METHOD CamAddPointToPath : BOOL
VAR_INPUT
	MotionFunctionFirstPoint : MC_MotionFunctionType;										  // Motion Function Type of initial Point in Cam Table. Start Postion is defined by current Positon of Axes.
	MotionFunctionThisPoint	 : MC_MotionFunctionType;										  // Motion Function Type of this Point to be added to Cam-Table
	PointNumber				 : UDINT(2..Parameter_Kinematic.MaxCammingPositionsPerTable);	  // Number of Point to be added to Cam Table, must be strictly increasing without gaps
	TotalPointsInTable		 : UDINT(2..Parameter_Kinematic.MaxCammingPositionsPerTable);	  // Total Number of Points in final Cam Table
	PointVelocity			 : ARRAY[1..KINEMATIC_CONSTANTS.DEGREES_OF_FREEDOM_MAX] OF LREAL; // Slave Velocity at this Point in Cam Table
	PointAcceleration		 : ARRAY[1..KINEMATIC_CONSTANTS.DEGREES_OF_FREEDOM_MAX] OF LREAL; // Slave Acceleration at this Point in Cam Table
	PointJerk				 : ARRAY[1..KINEMATIC_CONSTANTS.DEGREES_OF_FREEDOM_MAX] OF LREAL; // Slave Jerk at this Point in Cam Table
	PointIndex				 : UDINT;														  // Index of Point in structure of ST_BasePoint
END_VAR
IF _AcsAxesCam.CammingActive OR _McsAxesCam.CammingActive OR _AcsAxesCam.Busy OR _McsAxesCam.Busy THEN
	TRACE('CamAddPointToPath - Camming active or Buys');
	RETURN;
END_IF

IF SUPER^.KinematicStatus = E_KinStatus.KinStatus_Empty THEN
	CamAddPointToPath := _AcsAxesCam.CamAddPointToPath(MotionFunctionFirstPoint := MotionFunctionFirstPoint,
													   MotionFunctionThisPoint	:= MotionFunctionThisPoint,
													   PointNumber				:= PointNumber,
													   TotalPointsInTable		:= TotalPointsInTable,
													   Point					:= _CamPoints[PointIndex].AcsPosition,
													   PointVelocity			:= PointVelocity,
													   PointAcceleration		:= PointAcceleration,
													   PointJerk				:= PointJerk);
ELSIF SUPER^.KinematicStatus = E_KinStatus.KinStatus_Ready THEN
	CamAddPointToPath := _McsAxesCam.CamAddPointToPath(MotionFunctionFirstPoint := MotionFunctionFirstPoint,
													   MotionFunctionThisPoint	:= MotionFunctionThisPoint,
													   PointNumber				:= PointNumber,
													   TotalPointsInTable		:= TotalPointsInTable,
													   Point					:= _CamPoints[PointIndex].McsPosition,
													   PointVelocity			:= PointVelocity,
													   PointAcceleration		:= PointAcceleration,
													   PointJerk				:= PointJerk);
ELSE
	CamAddPointToPath := FALSE;
END_IF
END_METHOD

PROPERTY PUBLIC ChangeOccurred : BOOL
GET
ChangeOccurred := _ChangeOccurred;
END_GET
SET
_ChangeOccurred := ChangeOccurred;
END_SET
END_PROPERTY

METHOD PUBLIC GetPoint : ST_BasePoint
VAR_INPUT
	PointIndex : UDINT;
END_VAR
IF PointIndex > Parameter_Kinematic.MaxPoints THEN
	RETURN;
END_IF

GetPoint := _CamPoints[PointIndex];
END_METHOD

PROPERTY Points : REFERENCE TO ARRAY[0..Parameter_Kinematic.MaxPoints] OF ST_BasePoint
GET
Points REF= _CamPoints;
END_GET
END_PROPERTY

METHOD PUBLIC SetPoint : BOOL
VAR_INPUT
	Point	   : ST_BasePoint;
	PointIndex : UDINT;
END_VAR
IF PointIndex > Parameter_Kinematic.MaxPoints THEN
	RETURN;
END_IF

_CamPoints[PointIndex] := Point;
_ChangeOccurred		   := TRUE;
SetPoint			   := TRUE;
END_METHOD

PROPERTY CamInOptionsACS : ST_CamInOptions
GET
CamInOptionsACS := _AcsAxesCam.CamInOptions;
END_GET
SET
_AcsAxesCam.CamInOptions := CamInOptionsACS;
END_SET
END_PROPERTY

PROPERTY CamInOptionsMCS : ST_CamInOptions
GET
CamInOptionsMCS := _MCSAxesCam.CamInOptions;
END_GET
SET
_MCSAxesCam.CamInOptions := CamInOptionsMCS;
END_SET
END_PROPERTY

PROPERTY CamMasterAcs : REFERENCE TO AXIS_REF
GET
CamMasterAcs REF= _AcsAxesCam.CamMaster;
END_GET
END_PROPERTY

PROPERTY CamMasterMcs : REFERENCE TO AXIS_REF
GET
CamMasterMcs REF= _McsAxesCam.CamMaster;
END_GET
END_PROPERTY

PROPERTY CamTableSlaveDynamicsACS : ARRAY[1..KINEMATIC_CONSTANTS.DEGREES_OF_FREEDOM_MAX] OF ST_CamTableSlaveDynamics;
GET
CamTableSlaveDynamicsACS := _AcsAxesCam.CamTableSlaveDynamics;
END_GET
END_PROPERTY

PROPERTY CamTableSlaveDynamicsMCS : ARRAY[1..KINEMATIC_CONSTANTS.DEGREES_OF_FREEDOM_MAX] OF ST_CamTableSlaveDynamics;
GET
CamTableSlaveDynamicsMCS := _McsAxesCam.CamTableSlaveDynamics;
END_GET
END_PROPERTY

//! @summary Basic component initialization logic
METHOD PROTECTED Initialize : BOOL;
_AcsAxesCam.CamAxisCount := TO_UDINT(iAxis.AcsAxisCount);
_AcsAxesCam.CamAxisRef	 REF= iAxis.ACS;
_McsAxesCam.CamAxisCount := TO_UDINT(iAxis.DegreesOfFreedomConfigured);
_McsAxesCam.CamAxisRef	 REF= iAxis.MCS;
_AcsAxesCam.CyclicLogic(); // Init Run
_McsAxesCam.CyclicLogic(); // Init Run
IF SUPER^.Initialize() THEN
	Initialize := _AcsAxesCam.InitComplete AND _McsAxesCam.InitComplete;
END_IF
END_METHOD

END_FUNCTION_BLOCK

// Interfaces/I_KinematicCamming
INTERFACE I_KinematicCamming

METHOD CamClearPath : BOOL
VAR_INPUT
END_VAR
END_METHOD

METHOD CamIn : BOOL
VAR_INPUT
END_VAR
END_METHOD

METHOD CamMasterZero : BOOL
VAR_INPUT
END_VAR
END_METHOD

METHOD CamOut : BOOL
VAR_INPUT
END_VAR
END_METHOD

METHOD CamStartMovePath : BOOL
VAR_INPUT
	TargetMoveVelocity	   : LREAL := Parameter_Kinematic.CamDefaultMoveVelocity;	  // Move Velocity for Cam Table Master !!!Needs to consider all Slave dynamics, all Slaves try to follow Master setpoints!!!
	TargetMoveAcceleration : LREAL := Parameter_Kinematic.CamDefaultMoveAcceleration; // Move Acceleration for Cam Table Master !!!Needs to consider all Slave dynamics, all Slaves try to follow Master setpoints!!!
	TargetMoveDeceleration : LREAL := Parameter_Kinematic.CamDefaultMoveDeceleration; // Move Deceleration for Cam Table Master !!!Needs to consider all Slave dynamics, all Slaves try to follow Master setpoints!!!
	TargetMoveJerk		   : LREAL := Parameter_Kinematic.CamDefaultMoveJerk;		  // Move Jerk for Cam Table Master !!!Needs to consider all Slave dynamics, all Slaves try to follow Master setpoints!!!
END_VAR
END_METHOD

PROPERTY CammingActive : BOOL
GET
END_GET
END_PROPERTY

END_INTERFACE

// FunctionBlocks/FB_KinematicCamming
FUNCTION_BLOCK FB_KinematicCamming EXTENDS FB_CyclicFB IMPLEMENTS I_KinematicCamming
VAR
	// Kinematic Axis
	_CamVirtualMaster	  : AXIS_REF;
	_CamAxisRef			  : REFERENCE TO ARRAY[1..KINEMATIC_CONSTANTS.DEGREES_OF_FREEDOM_MAX] OF AXIS_REF;
	_CamAxisCount		  : UDINT := 1;
	_MotionFunctionPoints : ARRAY[1..KINEMATIC_CONSTANTS.DEGREES_OF_FREEDOM_MAX] OF UDINT(2..Parameter_Kinematic.MaxCammingPositionsPerTable) := [2,2,2,2,2,2];

	// Camming
	_McCamTableSelect		     : ARRAY[1..KINEMATIC_CONSTANTS.DEGREES_OF_FREEDOM_MAX] OF MC_CamTableSelect;
	_TableCamRef			     : ARRAY[1..KINEMATIC_CONSTANTS.DEGREES_OF_FREEDOM_MAX] OF MC_CAM_REF;
	_MotionFunctionPointsAxis1   : ARRAY[1..Parameter_Kinematic.MaxCammingPositionsPerTable] OF MC_MotionFunctionPoint;
	_MotionFunctionPointsAxis2   : ARRAY[1..Parameter_Kinematic.MaxCammingPositionsPerTable] OF MC_MotionFunctionPoint;
	_MotionFunctionPointsAxis3   : ARRAY[1..Parameter_Kinematic.MaxCammingPositionsPerTable] OF MC_MotionFunctionPoint;
	_MotionFunctionPointsAxis4   : ARRAY[1..Parameter_Kinematic.MaxCammingPositionsPerTable] OF MC_MotionFunctionPoint;
	_MotionFunctionPointsAxis5   : ARRAY[1..Parameter_Kinematic.MaxCammingPositionsPerTable] OF MC_MotionFunctionPoint;
	_MotionFunctionPointsAxis6   : ARRAY[1..Parameter_Kinematic.MaxCammingPositionsPerTable] OF MC_MotionFunctionPoint;
	_McCamIn				     : ARRAY[1..KINEMATIC_CONSTANTS.DEGREES_OF_FREEDOM_MAX] OF MC_CamIn;
	_McCamOut				     : ARRAY[1..KINEMATIC_CONSTANTS.DEGREES_OF_FREEDOM_MAX] OF MC_CamOut;
	_McReadCamTableSlaveDynamics : ARRAY[1..KINEMATIC_CONSTANTS.DEGREES_OF_FREEDOM_MAX] OF MC_ReadCamTableSlaveDynamics;
	_CamTableSlaveDynamics       : ARRAY[1..KINEMATIC_CONSTANTS.DEGREES_OF_FREEDOM_MAX] OF ST_CamTableSlaveDynamics;
	_McPowerVirtualMaster	     : MC_POWER;
	_McMoveAbs				     : MC_MoveAbsolute;
	_McHalt					     : MC_Halt;
	_McReset				     : MC_Reset;
	_McHome					     : MC_HOME;
	_CamInOptions                : ST_CamInOptions;

	// Internal Variables
	_KinematicCamInit		  : E_InitializeState_KinematicCamming := E_InitializeState_KinematicCamming.eInitializeState_Start;
	_i						  : UDINT;
	_MotionFunctionFirstPoint : MC_MotionFunctionType := MC_MotionFunctionType.MOTIONFUNCTYPE_POLYNOM5;
END_VAR

METHOD PUBLIC CyclicLogic
IF NOT _InitComplete THEN
	_InitComplete := THIS^.Initialize();
	RETURN;
END_IF

_CamVirtualMaster.ReadStatus();

(* Power Virtual Master *)
_McPowerVirtualMaster(Axis := _CamVirtualMaster, Enable_Positive := TRUE, Enable_Negative := TRUE);
IF _McPowerVirtualMaster.Error THEN
	_Error	 := TRUE;
	_ErrorId := _McPowerVirtualMaster.ErrorID;
END_IF

(* Reset Virtual Master *)
_McReset(Axis := _CamVirtualMaster);
IF _McReset.Error THEN
	_Error	 := TRUE;
	_ErrorId := _McReset.ErrorID;
END_IF

_McReset.Execute := FALSE;

(* Stop Virtual Master *)
_McHalt(Axis := _CamVirtualMaster);
IF _McHalt.Error THEN
	_Error	 := TRUE;
	_ErrorId := _McHalt.ErrorID;
END_IF

_McHalt.Execute := FALSE;

(* Move Virtual Master *)
_McMoveAbs(Axis := _CamVirtualMaster);
IF _McMoveAbs.Error THEN
	_Error	 := TRUE;
	_ErrorId := _McMoveAbs.ErrorID;
END_IF

_McMoveAbs.Execute := FALSE;

(* Reset Master to 0 *)
_McHome(Axis := _CamVirtualMaster, Position := 0.0, HomingMode := MC_HomingMOde.MC_Direct);
IF _McHome.Error THEN
	_Error	 := TRUE;
	_ErrorId := _McHome.ErrorID;
END_IF

_McHome.Execute := FALSE;

(* Reference Cam Table and initate first point *)
_TableCamRef[1].pArray		:= ADR(_MotionFunctionPointsAxis1);
_TableCamRef[1].ArraySize	:= SIZEOF(_MotionFunctionPointsAxis1);
_TableCamRef[1].TableType	:= MC_TableType.MC_TABLETYPE_MOTIONFUNCTION;
_TableCamRef[1].NoOfColumns := 1;
_TableCamRef[1].NoOfRows	:= _MotionFunctionPoints[1];
_TableCamRef[2].pArray		:= ADR(_MotionFunctionPointsAxis2);
_TableCamRef[2].ArraySize	:= SIZEOF(_MotionFunctionPointsAxis2);
_TableCamRef[2].TableType	:= MC_TableType.MC_TABLETYPE_MOTIONFUNCTION;
_TableCamRef[2].NoOfColumns := 1;
_TableCamRef[2].NoOfRows	:= _MotionFunctionPoints[2];
_TableCamRef[3].pArray		:= ADR(_MotionFunctionPointsAxis3);
_TableCamRef[3].ArraySize	:= SIZEOF(_MotionFunctionPointsAxis3);
_TableCamRef[3].TableType	:= MC_TableType.MC_TABLETYPE_MOTIONFUNCTION;
_TableCamRef[3].NoOfColumns := 1;
_TableCamRef[3].NoOfRows	:= _MotionFunctionPoints[3];
_TableCamRef[4].pArray		:= ADR(_MotionFunctionPointsAxis4);
_TableCamRef[4].ArraySize	:= SIZEOF(_MotionFunctionPointsAxis4);
_TableCamRef[4].TableType	:= MC_TableType.MC_TABLETYPE_MOTIONFUNCTION;
_TableCamRef[4].NoOfColumns := 1;
_TableCamRef[4].NoOfRows	:= _MotionFunctionPoints[4];
_TableCamRef[5].pArray		:= ADR(_MotionFunctionPointsAxis5);
_TableCamRef[5].ArraySize	:= SIZEOF(_MotionFunctionPointsAxis5);
_TableCamRef[5].TableType	:= MC_TableType.MC_TABLETYPE_MOTIONFUNCTION;
_TableCamRef[5].NoOfColumns := 1;
_TableCamRef[5].NoOfRows	:= _MotionFunctionPoints[5];
_TableCamRef[6].pArray		:= ADR(_MotionFunctionPointsAxis6);
_TableCamRef[6].ArraySize	:= SIZEOF(_MotionFunctionPointsAxis6);
_TableCamRef[6].TableType	:= MC_TableType.MC_TABLETYPE_MOTIONFUNCTION;
_TableCamRef[6].NoOfColumns := 1;
_TableCamRef[6].NoOfRows	:= _MotionFunctionPoints[6];
FOR _i := 1 TO _CamAxisCount DO
	(* Build Cam Table *)
	_McCamTableSelect[_i](Master		 := _CamVirtualMaster,
						  Slave			 := _CamAxisRef[_i],
						  CamTable		 := _TableCamRef[_i],
						  Periodic		 := Parameter_Kinematic.ExecuteCamPeriodically,
						  MasterAbsolute := Parameter_Kinematic.CamMasterAbsolute,
						  SlaveAbsolute	 := Parameter_Kinematic.CamSlaveAbsolute,
						  CamTableId	 := (_CamAxisRef[_i].NcToPlc.AxisId * 100));

	IF _McCamTableSelect[_i].Error THEN
		_Error	 := TRUE;
		_ErrorId := _McCamTableSelect[_i].ErrorID;
	END_IF

	_McCamTableSelect[_i].Execute := FALSE;

	(* Cam Axes to Master *)
	_McCamIn[_i](Master		   := _CamVirtualMaster,
				 Slave		   := _CamAxisRef[_i],
				 MasterOffset  := 0,
				 SlaveOffset   := 0,
				 MasterScaling := 1,
				 SlaveScaling  := 1,
				 StartMode	   := MC_STARTMODE.MC_STARTMODE_ABSOLUTE,
				 CamTableId	   := (_CamAxisRef[_i].NcToPlc.AxisId * 100),
				 Options	   := _CamInOptions);

	IF _McCamIn[_i].Error THEN
		_Error	 := TRUE;
		_ErrorId := _McCamIn[_i].ErrorID;
	END_IF

	_McCamIn[_i].Execute := FALSE;

	(* Cam Out Axes to Master *)
	_McCamOut[_i](Slave := _CamAxisRef[_i]);
	IF _McCamOut[_i].Error THEN
		_Error	 := TRUE;
		_ErrorId := _McCamOut[_i].ErrorID;
	END_IF

	_McCamOut[_i].Execute := FALSE;

	(* MC_ReadCamTableSlaveDynamics *)
	_McReadCamTableSlaveDynamics[_i](CamTableId		   := (_CamAxisRef[_i].NcToPlc.AxisId * 100),
									 SlavePosition	   => _CamTableSlaveDynamics[_i].SlavePosition,
									 SlaveVelocity	   => _CamTableSlaveDynamics[_i].SlaveVelocity,
									 SlaveAcceleration => _CamTableSlaveDynamics[_i].SlaveAcceleration);

	_McReadCamTableSlaveDynamics[_i].Execute := FALSE;
END_FOR

(* Create Busy Signal *)
_Busy := _McHalt.Busy OR _McReset.Busy OR _McMoveAbs.Busy OR _McHome.Busy;
FOR _i := 1 TO _CamAxisCount DO
	IF _McCamIn[_i].Busy OR _McCamOut[_i].Busy OR _McCamTableSelect[_i].Busy OR _McReadCamTableSlaveDynamics[_i].Busy THEN
		_Busy := TRUE;
	END_IF
END_FOR
END_METHOD

METHOD CamClearPath : BOOL
IF _Busy OR CammingActive THEN
	RETURN;
END_IF

MEMSET(destAddr := ADR(_MotionFunctionPointsAxis1), fillByte := 0, n := SIZEOF(_MotionFunctionPointsAxis1));
MEMSET(destAddr := ADR(_MotionFunctionPointsAxis2), fillByte := 0, n := SIZEOF(_MotionFunctionPointsAxis2));
MEMSET(destAddr := ADR(_MotionFunctionPointsAxis3), fillByte := 0, n := SIZEOF(_MotionFunctionPointsAxis3));
MEMSET(destAddr := ADR(_MotionFunctionPointsAxis4), fillByte := 0, n := SIZEOF(_MotionFunctionPointsAxis4));
MEMSET(destAddr := ADR(_MotionFunctionPointsAxis5), fillByte := 0, n := SIZEOF(_MotionFunctionPointsAxis5));
MEMSET(destAddr := ADR(_MotionFunctionPointsAxis6), fillByte := 0, n := SIZEOF(_MotionFunctionPointsAxis6));
CamClearPath := TRUE;
END_METHOD

METHOD CamIn : BOOL
IF _Busy OR CammingActive THEN
	RETURN;
END_IF

FOR _i := 1 TO _CamAxisCount DO
	_McCamIn[_i].Execute := TRUE;
END_FOR

CamIn := TRUE;
END_METHOD

METHOD CamMasterZero : BOOL
VAR_INPUT
END_VAR
IF _Busy OR CammingActive THEN
	RETURN;
END_IF

_McHome.Execute := TRUE;
CamMasterZero	:= TRUE;
END_METHOD

{attribute 'monitoring' := 'variable'}
PROPERTY CammingActive : BOOL
GET
CammingActive := TRUE;
FOR _i := 1 TO _CamAxisCount DO
	IF _CamAxisRef[_i].NcToPlc.CoupleState <> 3 THEN
		CammingActive := False;
	END_IF
END_FOR
END_GET
END_PROPERTY

METHOD CamOut : BOOL
IF _Busy THEN
	RETURN;
END_IF

FOR _i := 1 TO _CamAxisCount DO
	_McCamOut[_i].Execute := TRUE;
END_FOR

CamOut := TRUE;
END_METHOD

METHOD CamStartMovePath : BOOL
VAR_INPUT
	TargetMoveVelocity	   : LREAL := Parameter_Kinematic.CamDefaultMoveVelocity;	  // Move Velocity for Cam Table Master !!!Needs to consider all Slave dynamics, all Slaves try to follow Master setpoints!!!
	TargetMoveAcceleration : LREAL := Parameter_Kinematic.CamDefaultMoveAcceleration; // Move Acceleration for Cam Table Master !!!Needs to consider all Slave dynamics, all Slaves try to follow Master setpoints!!!
	TargetMoveDeceleration : LREAL := Parameter_Kinematic.CamDefaultMoveDeceleration; // Move Deceleration for Cam Table Master !!!Needs to consider all Slave dynamics, all Slaves try to follow Master setpoints!!!
	TargetMoveJerk		   : LREAL := Parameter_Kinematic.CamDefaultMoveJerk;		  // Move Jerk for Cam Table Master !!!Needs to consider all Slave dynamics, all Slaves try to follow Master setpoints!!!
END_VAR
IF _Busy OR NOT CammingActive THEN
	RETURN;
END_IF

_McMoveAbs.Jerk			:= TargetMoveJerk;
_McMoveAbs.Acceleration := TargetMoveAcceleration;
_McMoveAbs.Deceleration := TargetMoveDeceleration;
_McMoveAbs.Velocity		:= TargetMoveVelocity;
_McMoveAbs.Position		:= _CamVirtualMaster.NcToPlc.ActPos + 1.0;
_McMoveAbs.Execute		:= TRUE;
CamStartMovePath		:= TRUE;
END_METHOD

METHOD CamAddMotionPointByAxis : BOOL
VAR_INPUT
	Axis					 : UDINT(1..KINEMATIC_CONSTANTS.DEGREES_OF_FREEDOM_MAX);				   // Axis Number to add point to Cam table
	MotionFunctionFirstPoint : MC_MotionFunctionType := MC_MotionFunctionType.MOTIONFUNCTYPE_POLYNOM5; // Motion Function Type of initial Point in Cam Table. Start Postion is defined by current Positon of Axes.
	MotionFunctionThisPoint	 : MC_MotionFunctionType := MC_MotionFunctionType.MOTIONFUNCTYPE_POLYNOM5; // Motion Function Type of this Point to be added to Cam-Table
	PointNumber				 : UDINT(1..Parameter_Kinematic.MaxCammingPositionsPerTable);			   // Number of Point to be added to Cam Table, must be strictly increasing without gaps
	TotalPointsInTable		 : UDINT(2..Parameter_Kinematic.MaxCammingPositionsPerTable);			   // Total Number of Points in final Cam Table
	MasterPosition			 : LREAL;																   // Master Position for this Motion Point scaled to 1
	SlavePosition			 : LREAL;																   // Slave Position at this Point in Cam Table
	PointVelocity			 : LREAL;																   // Slave Velocity at this Point in Cam Table
	PointAcceleration		 : LREAL;																   // Slave Acceleration at this Point in Cam Table
	PointJerk				 : LREAL;																   // Slave Jerk at this Point in Cam Table
END_VAR

VAR
	_NextRelPoint : UDINT;
END_VAR
IF _Busy OR CammingActive THEN
	TRACE('CamAddMotionPointByAxis - Rejected buys or camming active!');
	RETURN;
END_IF

IF PointNumber > TotalPointsInTable OR PointNumber > Parameter_Kinematic.MaxCammingPositionsPerTable THEN
	TRACE('CamAddMotionPointByAxis - Rejected PointNumber invalid!');
	RETURN;
END_IF

IF MasterPosition < 0.0 OR MasterPosition > 1.0 THEN
	TRACE('CamAddMotionPointByAxis - Rejected MasterPosition not in allowed range of 0.0..1.0!');
	RETURN;
END_IF

IF NOT Parameter_Kinematic.CammingFirstPointInTableByUser THEN
	CamTableAddStartPoint();
END_IF

CASE Axis OF
	1:
		_MotionFunctionFirstPoint := MotionFunctionFirstPoint;
		IF PointNumber = TotalPointsInTable THEN
			_NextRelPoint				 := 0;
			_MotionFunctionPoints[1]	 := TotalPointsInTable;
			_McCamTableSelect[1].Execute := TRUE;
		ELSE
			_NextRelPoint := 1;
		END_IF

		_MotionFunctionPointsAxis1[PointNumber].PointIndex		  := PointNumber;
		_MotionFunctionPointsAxis1[PointNumber].FunctionType	  := MotionFunctionThisPoint;
		_MotionFunctionPointsAxis1[PointNumber].PointType		  := MC_MotionPointType.MOTIONPOINTTYPE_MOTION;
		_MotionFunctionPointsAxis1[PointNumber].MasterPos		  := MasterPosition;
		_MotionFunctionPointsAxis1[PointNumber].RelIndexNextPoint := _NextRelPoint;
		_MotionFunctionPointsAxis1[PointNumber].SlavePos		  := SlavePosition;
		_MotionFunctionPointsAxis1[PointNumber].SlaveVelo		  := PointVelocity;
		_MotionFunctionPointsAxis1[PointNumber].SlaveAcc		  := PointAcceleration;
		_MotionFunctionPointsAxis1[PointNumber].SlaveJerk		  := PointJerk;
		CamAddMotionPointByAxis									  := TRUE;

	2:
		_MotionFunctionFirstPoint := MotionFunctionFirstPoint;
		IF PointNumber = TotalPointsInTable THEN
			_NextRelPoint				 := 0;
			_MotionFunctionPoints[2]	 := TotalPointsInTable;
			_McCamTableSelect[2].Execute := TRUE;
		ELSE
			_NextRelPoint := 1;
		END_IF

		_MotionFunctionPointsAxis2[PointNumber].PointIndex		  := PointNumber;
		_MotionFunctionPointsAxis2[PointNumber].FunctionType	  := MotionFunctionThisPoint;
		_MotionFunctionPointsAxis2[PointNumber].PointType		  := MC_MotionPointType.MOTIONPOINTTYPE_MOTION;
		_MotionFunctionPointsAxis2[PointNumber].MasterPos		  := MasterPosition;
		_MotionFunctionPointsAxis2[PointNumber].RelIndexNextPoint := _NextRelPoint;
		_MotionFunctionPointsAxis2[PointNumber].SlavePos		  := SlavePosition;
		_MotionFunctionPointsAxis2[PointNumber].SlaveVelo		  := PointVelocity;
		_MotionFunctionPointsAxis2[PointNumber].SlaveAcc		  := PointAcceleration;
		_MotionFunctionPointsAxis2[PointNumber].SlaveJerk		  := PointJerk;
		CamAddMotionPointByAxis									  := TRUE;

	3:
		_MotionFunctionFirstPoint := MotionFunctionFirstPoint;
		IF PointNumber = TotalPointsInTable THEN
			_NextRelPoint				 := 0;
			_MotionFunctionPoints[3]	 := TotalPointsInTable;
			_McCamTableSelect[3].Execute := TRUE;
		ELSE
			_NextRelPoint := 1;
		END_IF

		_MotionFunctionPointsAxis3[PointNumber].PointIndex		  := PointNumber;
		_MotionFunctionPointsAxis3[PointNumber].FunctionType	  := MotionFunctionThisPoint;
		_MotionFunctionPointsAxis3[PointNumber].PointType		  := MC_MotionPointType.MOTIONPOINTTYPE_MOTION;
		_MotionFunctionPointsAxis3[PointNumber].MasterPos		  := MasterPosition;
		_MotionFunctionPointsAxis3[PointNumber].RelIndexNextPoint := _NextRelPoint;
		_MotionFunctionPointsAxis3[PointNumber].SlavePos		  := SlavePosition;
		_MotionFunctionPointsAxis3[PointNumber].SlaveVelo		  := PointVelocity;
		_MotionFunctionPointsAxis3[PointNumber].SlaveAcc		  := PointAcceleration;
		_MotionFunctionPointsAxis3[PointNumber].SlaveJerk		  := PointJerk;
		CamAddMotionPointByAxis									  := TRUE;

	4:
		_MotionFunctionFirstPoint := MotionFunctionFirstPoint;
		IF PointNumber = TotalPointsInTable THEN
			_NextRelPoint				 := 0;
			_MotionFunctionPoints[4]	 := TotalPointsInTable;
			_McCamTableSelect[4].Execute := TRUE;
		ELSE
			_NextRelPoint := 1;
		END_IF

		_MotionFunctionPointsAxis4[PointNumber].PointIndex		  := PointNumber;
		_MotionFunctionPointsAxis4[PointNumber].FunctionType	  := MotionFunctionThisPoint;
		_MotionFunctionPointsAxis4[PointNumber].PointType		  := MC_MotionPointType.MOTIONPOINTTYPE_MOTION;
		_MotionFunctionPointsAxis4[PointNumber].MasterPos		  := MasterPosition;
		_MotionFunctionPointsAxis4[PointNumber].RelIndexNextPoint := _NextRelPoint;
		_MotionFunctionPointsAxis4[PointNumber].SlavePos		  := SlavePosition;
		_MotionFunctionPointsAxis4[PointNumber].SlaveVelo		  := PointVelocity;
		_MotionFunctionPointsAxis4[PointNumber].SlaveAcc		  := PointAcceleration;
		_MotionFunctionPointsAxis4[PointNumber].SlaveJerk		  := PointJerk;
		CamAddMotionPointByAxis									  := TRUE;

	5:
		_MotionFunctionFirstPoint := MotionFunctionFirstPoint;
		IF PointNumber = TotalPointsInTable THEN
			_NextRelPoint				 := 0;
			_MotionFunctionPoints[5]	 := TotalPointsInTable;
			_McCamTableSelect[5].Execute := TRUE;
		ELSE
			_NextRelPoint := 1;
		END_IF

		_MotionFunctionPointsAxis5[PointNumber].PointIndex		  := PointNumber;
		_MotionFunctionPointsAxis5[PointNumber].FunctionType	  := MotionFunctionThisPoint;
		_MotionFunctionPointsAxis5[PointNumber].PointType		  := MC_MotionPointType.MOTIONPOINTTYPE_MOTION;
		_MotionFunctionPointsAxis5[PointNumber].MasterPos		  := MasterPosition;
		_MotionFunctionPointsAxis5[PointNumber].RelIndexNextPoint := _NextRelPoint;
		_MotionFunctionPointsAxis5[PointNumber].SlavePos		  := SlavePosition;
		_MotionFunctionPointsAxis5[PointNumber].SlaveVelo		  := PointVelocity;
		_MotionFunctionPointsAxis5[PointNumber].SlaveAcc		  := PointAcceleration;
		_MotionFunctionPointsAxis5[PointNumber].SlaveJerk		  := PointJerk;
		CamAddMotionPointByAxis									  := TRUE;

	6:
		_MotionFunctionFirstPoint := MotionFunctionFirstPoint;
		IF PointNumber = TotalPointsInTable THEN
			_NextRelPoint				 := 0;
			_MotionFunctionPoints[6]	 := TotalPointsInTable;
			_McCamTableSelect[6].Execute := TRUE;
		ELSE
			_NextRelPoint := 1;
		END_IF

		_MotionFunctionPointsAxis6[PointNumber].PointIndex		  := PointNumber;
		_MotionFunctionPointsAxis6[PointNumber].FunctionType	  := MotionFunctionThisPoint;
		_MotionFunctionPointsAxis6[PointNumber].PointType		  := MC_MotionPointType.MOTIONPOINTTYPE_MOTION;
		_MotionFunctionPointsAxis6[PointNumber].MasterPos		  := MasterPosition;
		_MotionFunctionPointsAxis6[PointNumber].RelIndexNextPoint := _NextRelPoint;
		_MotionFunctionPointsAxis6[PointNumber].SlavePos		  := SlavePosition;
		_MotionFunctionPointsAxis6[PointNumber].SlaveVelo		  := PointVelocity;
		_MotionFunctionPointsAxis6[PointNumber].SlaveAcc		  := PointAcceleration;
		_MotionFunctionPointsAxis6[PointNumber].SlaveJerk		  := PointJerk;
		CamAddMotionPointByAxis									  := TRUE;

ELSE
	TRACE('CamAddMotionPointByAxis - Rejected Axis number not valid');
END_CASE
END_METHOD

METHOD CamAddPointToPath : BOOL
VAR_INPUT
	MotionFunctionFirstPoint : MC_MotionFunctionType := MC_MotionFunctionType.MOTIONFUNCTYPE_POLYNOM5; // Motion Function Type of initial Point in Cam Table. Start Postion is defined by current Positon of Axes.
	MotionFunctionThisPoint	 : MC_MotionFunctionType := MC_MotionFunctionType.MOTIONFUNCTYPE_POLYNOM5; // Motion Function Type of this Point to be added to Cam-Table
	PointNumber				 : UDINT(2..Parameter_Kinematic.MaxCammingPositionsPerTable);			   // Number of Point to be added to Cam Table, must be strictly increasing without gaps
	TotalPointsInTable		 : UDINT(2..Parameter_Kinematic.MaxCammingPositionsPerTable);			   // Total Number of Points in final Cam Table
	Point					 : ARRAY[1..KINEMATIC_CONSTANTS.DEGREES_OF_FREEDOM_MAX] OF LREAL;		   // Slave Position at this Point in Cam Table
	PointVelocity			 : ARRAY[1..KINEMATIC_CONSTANTS.DEGREES_OF_FREEDOM_MAX] OF LREAL;		   // Slave Velocity at this Point in Cam Table
	PointAcceleration		 : ARRAY[1..KINEMATIC_CONSTANTS.DEGREES_OF_FREEDOM_MAX] OF LREAL;		   // Slave Acceleration at this Point in Cam Table
	PointJerk				 : ARRAY[1..KINEMATIC_CONSTANTS.DEGREES_OF_FREEDOM_MAX] OF LREAL;		   // Slave Jerk at this Point in Cam Table
END_VAR

VAR
	_NextRelPoint : UDINT;
END_VAR
IF _Busy OR CammingActive THEN
	TRACE('CamAddPointToPath - Rejected buys or camming active!');
	RETURN;
END_IF

IF PointNumber > TotalPointsInTable OR PointNumber > Parameter_Kinematic.MaxCammingPositionsPerTable THEN
	TRACE('CamAddPointToPath - Rejected PointNumber invalid!');
	RETURN;
END_IF

_MotionFunctionFirstPoint := MotionFunctionFirstPoint;
IF PointNumber = TotalPointsInTable THEN
	_NextRelPoint := 0;
	CamTableAddStartPoint();
	FOR _i := 1 TO _CamAxisCount DO
		_MotionFunctionPoints[_i]	  := TotalPointsInTable;
		_McCamTableSelect[_i].Execute := TRUE;
	END_FOR
ELSE
	_NextRelPoint := 1;
END_IF

_MotionFunctionPointsAxis1[PointNumber].PointIndex		  := PointNumber;
_MotionFunctionPointsAxis1[PointNumber].FunctionType	  := MotionFunctionThisPoint;
_MotionFunctionPointsAxis1[PointNumber].PointType		  := MC_MotionPointType.MOTIONPOINTTYPE_MOTION;
_MotionFunctionPointsAxis1[PointNumber].MasterPos		  := _CamVirtualMaster.NcToPlc.ActPos + ((1.0 / TO_REAL(TotalPointsInTable) * TO_REAL(PointNumber)));
_MotionFunctionPointsAxis1[PointNumber].RelIndexNextPoint := _NextRelPoint;
_MotionFunctionPointsAxis1[PointNumber].SlavePos		  := Point[1];
_MotionFunctionPointsAxis1[PointNumber].SlaveVelo		  := PointVelocity[1];
_MotionFunctionPointsAxis1[PointNumber].SlaveAcc		  := PointAcceleration[1];
_MotionFunctionPointsAxis1[PointNumber].SlaveJerk		  := PointJerk[1];
_MotionFunctionPointsAxis2[PointNumber].PointIndex		  := PointNumber;
_MotionFunctionPointsAxis2[PointNumber].FunctionType	  := MotionFunctionThisPoint;
_MotionFunctionPointsAxis2[PointNumber].PointType		  := MC_MotionPointType.MOTIONPOINTTYPE_MOTION;
_MotionFunctionPointsAxis2[PointNumber].MasterPos		  := _CamVirtualMaster.NcToPlc.ActPos + ((1.0 / TO_REAL(TotalPointsInTable) * TO_REAL(PointNumber)));
_MotionFunctionPointsAxis2[PointNumber].RelIndexNextPoint := _NextRelPoint;
_MotionFunctionPointsAxis2[PointNumber].SlavePos		  := Point[2];
_MotionFunctionPointsAxis2[PointNumber].SlaveVelo		  := PointVelocity[2];
_MotionFunctionPointsAxis2[PointNumber].SlaveAcc		  := PointAcceleration[2];
_MotionFunctionPointsAxis2[PointNumber].SlaveJerk		  := PointJerk[2];
_MotionFunctionPointsAxis3[PointNumber].PointIndex		  := PointNumber;
_MotionFunctionPointsAxis3[PointNumber].FunctionType	  := MotionFunctionThisPoint;
_MotionFunctionPointsAxis3[PointNumber].PointType		  := MC_MotionPointType.MOTIONPOINTTYPE_MOTION;
_MotionFunctionPointsAxis3[PointNumber].MasterPos		  := _CamVirtualMaster.NcToPlc.ActPos + ((1.0 / TO_REAL(TotalPointsInTable) * TO_REAL(PointNumber)));
_MotionFunctionPointsAxis3[PointNumber].RelIndexNextPoint := _NextRelPoint;
_MotionFunctionPointsAxis3[PointNumber].SlavePos		  := Point[3];
_MotionFunctionPointsAxis3[PointNumber].SlaveVelo		  := PointVelocity[3];
_MotionFunctionPointsAxis3[PointNumber].SlaveAcc		  := PointAcceleration[3];
_MotionFunctionPointsAxis3[PointNumber].SlaveJerk		  := PointJerk[3];
_MotionFunctionPointsAxis4[PointNumber].PointIndex		  := PointNumber;
_MotionFunctionPointsAxis4[PointNumber].FunctionType	  := MotionFunctionThisPoint;
_MotionFunctionPointsAxis4[PointNumber].PointType		  := MC_MotionPointType.MOTIONPOINTTYPE_MOTION;
_MotionFunctionPointsAxis4[PointNumber].MasterPos		  := _CamVirtualMaster.NcToPlc.ActPos + ((1.0 / TO_REAL(TotalPointsInTable) * TO_REAL(PointNumber)));
_MotionFunctionPointsAxis4[PointNumber].RelIndexNextPoint := _NextRelPoint;
_MotionFunctionPointsAxis4[PointNumber].SlavePos		  := Point[4];
_MotionFunctionPointsAxis4[PointNumber].SlaveVelo		  := PointVelocity[4];
_MotionFunctionPointsAxis4[PointNumber].SlaveAcc		  := PointAcceleration[4];
_MotionFunctionPointsAxis4[PointNumber].SlaveJerk		  := PointJerk[4];
_MotionFunctionPointsAxis5[PointNumber].PointIndex		  := PointNumber;
_MotionFunctionPointsAxis5[PointNumber].FunctionType	  := MotionFunctionThisPoint;
_MotionFunctionPointsAxis5[PointNumber].PointType		  := MC_MotionPointType.MOTIONPOINTTYPE_MOTION;
_MotionFunctionPointsAxis5[PointNumber].MasterPos		  := _CamVirtualMaster.NcToPlc.ActPos + ((1.0 / TO_REAL(TotalPointsInTable) * TO_REAL(PointNumber)));
_MotionFunctionPointsAxis5[PointNumber].RelIndexNextPoint := _NextRelPoint;
_MotionFunctionPointsAxis5[PointNumber].SlavePos		  := Point[5];
_MotionFunctionPointsAxis5[PointNumber].SlaveVelo		  := PointVelocity[5];
_MotionFunctionPointsAxis5[PointNumber].SlaveAcc		  := PointAcceleration[5];
_MotionFunctionPointsAxis5[PointNumber].SlaveJerk		  := PointJerk[5];
_MotionFunctionPointsAxis6[PointNumber].PointIndex		  := PointNumber;
_MotionFunctionPointsAxis6[PointNumber].FunctionType	  := MotionFunctionThisPoint;
_MotionFunctionPointsAxis6[PointNumber].PointType		  := MC_MotionPointType.MOTIONPOINTTYPE_MOTION;
_MotionFunctionPointsAxis6[PointNumber].MasterPos		  := _CamVirtualMaster.NcToPlc.ActPos + ((1.0 / TO_REAL(TotalPointsInTable) * TO_REAL(PointNumber)));
_MotionFunctionPointsAxis6[PointNumber].RelIndexNextPoint := _NextRelPoint;
_MotionFunctionPointsAxis6[PointNumber].SlavePos		  := Point[6];
_MotionFunctionPointsAxis6[PointNumber].SlaveVelo		  := PointVelocity[6];
_MotionFunctionPointsAxis6[PointNumber].SlaveAcc		  := PointAcceleration[6];
_MotionFunctionPointsAxis6[PointNumber].SlaveJerk		  := PointJerk[6];
CamAddPointToPath										  := TRUE;
END_METHOD

METHOD PRIVATE CamTableAddStartPoint
VAR_INPUT
END_VAR
//
_MotionFunctionPointsAxis1[1].PointIndex		:= 1;
_MotionFunctionPointsAxis1[1].FunctionType		:= _MotionFunctionFirstPoint;
_MotionFunctionPointsAxis1[1].PointType			:= MC_MotionPointType.MOTIONPOINTTYPE_MOTION;
_MotionFunctionPointsAxis1[1].RelIndexNextPoint := 1;
_MotionFunctionPointsAxis1[1].MasterPos			:= _CamVirtualMaster.NcToPlc.ActPos;
_MotionFunctionPointsAxis1[1].SlavePos			:= _CamAxisRef[1].NcToPlc.ActPos;
_MotionFunctionPointsAxis1[1].SlaveVelo			:= 0;
_MotionFunctionPointsAxis1[1].SlaveAcc			:= 0;
_MotionFunctionPointsAxis1[1].SlaveJerk			:= 0;

//
_MotionFunctionPointsAxis2[1].PointIndex		:= 1;
_MotionFunctionPointsAxis2[1].FunctionType		:= _MotionFunctionFirstPoint;
_MotionFunctionPointsAxis2[1].PointType			:= MC_MotionPointType.MOTIONPOINTTYPE_MOTION;
_MotionFunctionPointsAxis2[1].RelIndexNextPoint := 1;
_MotionFunctionPointsAxis2[1].MasterPos			:= _CamVirtualMaster.NcToPlc.ActPos;
_MotionFunctionPointsAxis2[1].SlavePos			:= _CamAxisRef[2].NcToPlc.ActPos;
_MotionFunctionPointsAxis2[1].SlaveVelo			:= 0;
_MotionFunctionPointsAxis2[1].SlaveAcc			:= 0;
_MotionFunctionPointsAxis2[1].SlaveJerk			:= 0;

//
_MotionFunctionPointsAxis3[1].PointIndex		:= 1;
_MotionFunctionPointsAxis3[1].FunctionType		:= _MotionFunctionFirstPoint;
_MotionFunctionPointsAxis3[1].PointType			:= MC_MotionPointType.MOTIONPOINTTYPE_MOTION;
_MotionFunctionPointsAxis3[1].RelIndexNextPoint := 1;
_MotionFunctionPointsAxis3[1].MasterPos			:= _CamVirtualMaster.NcToPlc.ActPos;
_MotionFunctionPointsAxis3[1].SlavePos			:= _CamAxisRef[3].NcToPlc.ActPos;
_MotionFunctionPointsAxis3[1].SlaveVelo			:= 0;
_MotionFunctionPointsAxis3[1].SlaveAcc			:= 0;
_MotionFunctionPointsAxis3[1].SlaveJerk			:= 0;

//
_MotionFunctionPointsAxis4[1].PointIndex		:= 1;
_MotionFunctionPointsAxis4[1].FunctionType		:= _MotionFunctionFirstPoint;
_MotionFunctionPointsAxis4[1].PointType			:= MC_MotionPointType.MOTIONPOINTTYPE_MOTION;
_MotionFunctionPointsAxis4[1].RelIndexNextPoint := 1;
_MotionFunctionPointsAxis4[1].MasterPos			:= _CamVirtualMaster.NcToPlc.ActPos;
_MotionFunctionPointsAxis4[1].SlavePos			:= _CamAxisRef[4].NcToPlc.ActPos;
_MotionFunctionPointsAxis4[1].SlaveVelo			:= 0;
_MotionFunctionPointsAxis4[1].SlaveAcc			:= 0;
_MotionFunctionPointsAxis4[1].SlaveJerk			:= 0;

//
_MotionFunctionPointsAxis5[1].PointIndex		:= 1;
_MotionFunctionPointsAxis5[1].FunctionType		:= _MotionFunctionFirstPoint;
_MotionFunctionPointsAxis5[1].PointType			:= MC_MotionPointType.MOTIONPOINTTYPE_MOTION;
_MotionFunctionPointsAxis5[1].RelIndexNextPoint := 1;
_MotionFunctionPointsAxis5[1].MasterPos			:= _CamVirtualMaster.NcToPlc.ActPos;
_MotionFunctionPointsAxis5[1].SlavePos			:= _CamAxisRef[5].NcToPlc.ActPos;
_MotionFunctionPointsAxis5[1].SlaveVelo			:= 0;
_MotionFunctionPointsAxis5[1].SlaveAcc			:= 0;
_MotionFunctionPointsAxis5[1].SlaveJerk			:= 0;

//
_MotionFunctionPointsAxis6[1].PointIndex		:= 1;
_MotionFunctionPointsAxis6[1].FunctionType		:= _MotionFunctionFirstPoint;
_MotionFunctionPointsAxis6[1].PointType			:= MC_MotionPointType.MOTIONPOINTTYPE_MOTION;
_MotionFunctionPointsAxis6[1].RelIndexNextPoint := 1;
_MotionFunctionPointsAxis6[1].MasterPos			:= _CamVirtualMaster.NcToPlc.ActPos;
_MotionFunctionPointsAxis6[1].SlavePos			:= _CamAxisRef[6].NcToPlc.ActPos;
_MotionFunctionPointsAxis6[1].SlaveVelo			:= 0;
_MotionFunctionPointsAxis6[1].SlaveAcc			:= 0;
_MotionFunctionPointsAxis6[1].SlaveJerk			:= 0;
END_METHOD

METHOD Disable : BOOL
VAR_INPUT
END_VAR
_McPowerVirtualMaster.Enable := FALSE;
Disable						 := TRUE;
END_METHOD

METHOD Enable : BOOL
VAR_INPUT
END_VAR
_McPowerVirtualMaster.Enable := TRUE;
Enable						 := TRUE;
END_METHOD

METHOD ReadCamTableSlaveDynamics : BOOL // Results of read in Property CamTableSlaveDynamics
VAR_INPUT
	MasterPosition : LREAL;
END_VAR
FOR _i := 1 TO _CamAxisCount DO
	_McReadCamTableSlaveDynamics[_i].MasterPosition := MasterPosition;
	_McReadCamTableSlaveDynamics[_i].Execute		:= TRUE;
END_FOR

ReadCamTableSlaveDynamics := TRUE;
END_METHOD

METHOD Reset : BOOL
VAR_INPUT
END_VAR
_McReset.Execute := TRUE;
_Error			 := FALSE;
_ErrorId		 := 0;
Reset			 := TRUE;
END_METHOD

METHOD SetOverride : BOOL
VAR_INPUT
	Override : LREAL := 100.0; // 100.0 = 100% Full Speed
END_VAR
_McPowerVirtualMaster.Override := Override;
SetOverride					   := TRUE;
END_METHOD

METHOD Stop : BOOL
VAR_INPUT
	Deceleration : LREAL;
	Jerk		 : LREAL;
END_VAR
IF Deceleration = 0 OR Jerk = 0 THEN
	_McHalt.Deceleration := Parameter_Kinematic.DefaultStopDeceleration;
	_McHalt.Jerk		 := Parameter_Kinematic.DefaultStopDecelerationJerk;
ELSE
	_McHalt.Deceleration := Deceleration;
	_McHalt.Jerk		 := Jerk;
END_IF

_McHalt.Execute := TRUE;
Stop			:= TRUE;
END_METHOD

{attribute 'monitoring' := 'variable'}
PROPERTY Public CamAxisCount : UDINT
SET
_CamAxisCount := CamAxisCount;
END_SET
END_PROPERTY

PROPERTY CamAxisRef : REFERENCE TO ARRAY[1..KINEMATIC_CONSTANTS.DEGREES_OF_FREEDOM_MAX] OF AXIS_REF
GET
CamAxisRef REf= _CamAxisRef;
END_GET
SET
_CamAxisRef REF= CamAxisRef;
END_SET
END_PROPERTY

PROPERTY CamInOptions : ST_CamInOptions
GET
CamInOptions := _CamInOptions;
END_GET
SET
_CamInOptions := CamInOptions;
END_SET
END_PROPERTY

PROPERTY CamMaster : REFERENCE TO AXIS_REF
GET
CamMaster REF= _CamVirtualMaster;
END_GET
END_PROPERTY

PROPERTY CamTableSlaveDynamics : ARRAY[1..KINEMATIC_CONSTANTS.DEGREES_OF_FREEDOM_MAX] OF ST_CamTableSlaveDynamics;
GET
CamTableSlaveDynamics := _CamTableSlaveDynamics;
END_GET
END_PROPERTY

METHOD Initialize : BOOL
VAR_INPUT
END_VAR
CASE _KinematicCamInit OF
	E_InitializeState_KinematicCamming.eInitializeState_Start:
		Initialize := FALSE;
		IF _CamAxisCount > 6 THEN
			TRACE('Too many Axes connected to Camming FB! Only up to DOF=6 possible!');
			_KinematicCamInit := E_InitializeState_KinematicCamming.eInitializeState_Failed;
			RETURN;
		ELSE
			_KinematicCamInit := E_InitializeState_KinematicCamming.eInitializeState_CheckLinking;
		END_IF

	E_InitializeState_KinematicCamming.eInitializeState_CheckLinking:
		IF F_GetMappingStatus(ADR(_CamVirtualMaster.NcToPlc), SIZEOF(_CamVirtualMaster.NcToPlc)) <> EPlcMappingStatus.MS_Mapped OR F_GetMappingStatus(ADR(_CamVirtualMaster.PlcToNc), SIZEOF(_CamVirtualMaster.PlcToNc)) <> EPlcMappingStatus.MS_Mapped THEN
			Trace('Programming Error init failed with Virtual Camming Master Axis Link missing!');
			_KinematicCamInit := E_InitializeState_KinematicCamming.eInitializeState_Failed;
		ELSE
			_KinematicCamInit := E_InitializeState_KinematicCamming.eInitializeState_CheckRef;
		END_IF

	E_InitializeState_KinematicCamming.eInitializeState_CheckRef:
		IF NOT __ISVALIDREF(_CamAxisRef) THEN
			Trace('Programming Error init failed Axes System not referenced!');
			_KinematicCamInit := E_InitializeState_KinematicCamming.eInitializeState_Failed;
		ELSE
			_KinematicCamInit := E_InitializeState_KinematicCamming.eInitializeState_Done;
		END_IF

	E_InitializeState_KinematicCamming.eInitializeState_Done:
		_Busy	   := FALSE;
		Initialize := TRUE;

	E_InitializeState_KinematicCamming.eInitializeState_Failed:
		_Busy  := FALSE;
		_Error := TRUE;
END_CASE
END_METHOD

END_FUNCTION_BLOCK

// FunctionBlocks/FB_KinematicAxisRef
FUNCTION_BLOCK FB_KinematicAxisRef IMPLEMENTS I_KinematicAxisRef
VAR
	AcsAxis						: ARRAY[1..KINEMATIC_CONSTANTS.DEGREES_OF_FREEDOM_MAX] OF AXIS_REF;
	McsAxis						: ARRAY[1..KINEMATIC_CONSTANTS.DEGREES_OF_FREEDOM_MAX] OF AXIS_REF;
	_DegreesOfFreedomConfigured : E_KinematicDOF := E_KinematicDOF.eKinematicDOF_Max; // MCS
	_AcsAxisCount				: UDINT;											  // ACS
	_AcsPositionAbsolute		: BOOL;
END_VAR

PROPERTY ACS : REFERENCE TO ARRAY[1..KINEMATIC_CONSTANTS.DEGREES_OF_FREEDOM_MAX] OF AXIS_REF
GET
ACS REF= AcsAxis;
END_GET
END_PROPERTY

PROPERTY AcsAxisCount : UDINT
GET
AcsAxisCount := _AcsAxisCount;
END_GET
SET
_AcsAxisCount := AcsAxisCount;
END_SET
END_PROPERTY

PROPERTY AcsPositionAbsolute : BOOL
GET
AcsPositionAbsolute := _AcsPositionAbsolute;
END_GET
SET
_AcsPositionAbsolute := AcsPositionAbsolute;
END_SET
END_PROPERTY

{attribute 'monitoring' := 'variable'}
PROPERTY DegreesOfFreedomConfigured : E_KinematicDOF
GET
DegreesOfFreedomConfigured := _DegreesOfFreedomConfigured;
END_GET
SET
_DegreesOfFreedomConfigured := DegreesOfFreedomConfigured;
END_SET
END_PROPERTY

PROPERTY MCS : REFERENCE TO ARRAY[1..KINEMATIC_CONSTANTS.DEGREES_OF_FREEDOM_MAX] OF AXIS_REF
GET
MCS REF= McsAxis;
END_GET
END_PROPERTY

END_FUNCTION_BLOCK

// Project Information/F_GetCompany
// This function has been automatically generated from the project information.
{attribute 'signature_flag' := '1073741824'}
{attribute 'TcGenerated'}
{attribute 'no-analysis'}
FUNCTION F_GetCompany : WSTRING
VAR_INPUT
	
END_VAR

F_GetCompany := "Beckhoff Automation LLC";

END_FUNCTION

// Project Information/F_GetTitle
// This function has been automatically generated from the project information.
{attribute 'signature_flag' := '1073741824'}
{attribute 'TcGenerated'}
{attribute 'no-analysis'}
FUNCTION F_GetTitle : WSTRING
VAR_INPUT
	
END_VAR

F_GetTitle := "SPT Kinematics";

END_FUNCTION

// Project Information/F_GetVersion
// This function has been automatically generated from the project information.
{attribute 'signature_flag' := '1073741824'}
{attribute 'TcGenerated'}
{attribute 'no-analysis'}
FUNCTION F_GetVersion : ST_LibVersion
VAR_INPUT
	
END_VAR

F_GetVersion.iMajor := 3;
F_GetVersion.iMinor := 3;
F_GetVersion.iBuild := 5;
F_GetVersion.iRevision := 0;
F_GetVersion.sVersion := '3.3.5';
F_GetVersion.nFlags := 1;

END_FUNCTION
